LIN {X 0,Y 63.394,Z 649.51,A -85,B 0,C 180,E1 -25836.083,E2 -25836.083} C_VEL
LIN {X 0,Y 63.785,Z 649.473,A -85,B 0,C 180,E1 -25829.999,E2 -25829.999} C_VEL
LIN {X 0,Y 63.352,Z 649.516,A -85,B 0,C 180,E1 -25823.651,E2 -25823.651} C_VEL
LIN {X 0,Y 62.733,Z 649.594,A -85,B 0,C 180,E1 -25817.095,E2 -25817.095} C_VEL
LIN {X 0,Y 62.53,Z 649.629,A -85,B 0,C 180,E1 -25810.362,E2 -25810.362} C_VEL
LIN {X 0,Y 62.407,Z 649.638,A -85,B 0,C 180,E1 -25803.322,E2 -25803.322} C_VEL
LIN {X 0,Y 62.272,Z 649.648,A -85,B 0,C 180,E1 -25795.776,E2 -25795.776} C_VEL
LIN {X 0,Y 62.265,Z 649.651,A -85,B 0,C 180,E1 -25787.547,E2 -25787.547} C_VEL
LIN {X 0,Y 62.489,Z 649.625,A -85,B 0,C 180,E1 -25778.311,E2 -25778.311} C_VEL
LIN {X 0,Y 63.859,Z 649.453,A -85,B 0,C 180,E1 -25766.021,E2 -25766.021} C_VEL
LIN {X 0,Y 67.059,Z 649.057,A -85,B 0,C 180,E1 -25755.851,E2 -25755.851} C_VEL
LIN {X 0,Y 69.864,Z 669.968,A -85,B 0,C 180,E1 -25752.483,E2 -25752.483} C_VEL
LIN {X 0,Y 73.414,Z 727.269,A -85,B 0,C 180,E1 -25741.194,E2 -25741.194} C_VEL
LIN {X 0,Y 74.444,Z 742.789,A -85,B 0,C 180,E1 -25737.808,E2 -25737.808} C_VEL
LIN {X 0,Y 75.346,Z 754.304,A -85,B 0,C 180,E1 -25734.33,E2 -25734.33} C_VEL
LIN {X 0,Y 76.271,Z 762.21,A -85,B 0,C 180,E1 -25731.416,E2 -25731.416} C_VEL
LIN {X 0,Y 77.368,Z 770.599,A -85,B 0,C 180,E1 -25727.582,E2 -25727.582} C_VEL
LIN {X 0,Y 78.462,Z 778.205,A -85,B 0,C 180,E1 -25723.132,E2 -25723.132} C_VEL
LIN {X 0,Y 81.222,Z 788.982,A -85,B 0,C 180,E1 -25715.817,E2 -25715.817} C_VEL
LIN {X 0,Y 86.34,Z 799.372,A -85,B 0,C 180,E1 -25708.174,E2 -25708.174} C_VEL
LIN {X 0,Y 93.196,Z 808.561,A -85,B 0,C 180,E1 -25701.678,E2 -25701.678} C_VEL
LIN {X 0,Y 94.313,Z 809.773,A -85,B 0,C 180,E1 -25700.854,E2 -25700.854} C_VEL
LIN {X 0,Y 94.62,Z 810.111,A -85,B 0,C 180,E1 -25699.452,E2 -25699.452} C_VEL
LIN {X 0,Y 88.677,Z 803.193,A -85,B 0,C 180,E1 -25693.883,E2 -25693.883} C_VEL
LIN {X 0,Y 84.114,Z 795.657,A -85,B 0,C 180,E1 -25687.442,E2 -25687.442} C_VEL
LIN {X 0,Y 81.243,Z 787.247,A -85,B 0,C 180,E1 -25680.438,E2 -25680.438} C_VEL
LIN {X 0,Y 80.047,Z 778.623,A -85,B 0,C 180,E1 -25673.713,E2 -25673.713} C_VEL
LIN {X 0,Y 78.629,Z 771.489,A -85,B 0,C 180,E1 -25670.195,E2 -25670.195} C_VEL
LIN {X 0,Y 76.861,Z 760.414,A -85,B 0,C 180,E1 -25665.867,E2 -25665.867} C_VEL
LIN {X 0,Y 75.569,Z 748.02,A -85,B 0,C 180,E1 -25662.208,E2 -25662.208} C_VEL
LIN {X 0,Y 74.133,Z 730.465,A -85,B 0,C 180,E1 -25658.491,E2 -25658.491} C_VEL
LIN {X 0,Y 71.014,Z 689.149,A -85,B 0,C 180,E1 -25650.599,E2 -25650.599} C_VEL
LIN {X 0,Y 66.636,Z 656.391,A -85,B 0,C 180,E1 -25645.481,E2 -25645.481} C_VEL
LIN {X 0,Y 65.955,Z 649.201,A -85,B 0,C 180,E1 -25644.096,E2 -25644.096} C_VEL
LIN {X 0,Y 62.604,Z 649.615,A -85,B 0,C 180,E1 -25623.415,E2 -25623.415} C_VEL
LIN {X 0,Y 62.375,Z 649.648,A -85,B 0,C 180,E1 -25615.843,E2 -25615.843} C_VEL
LIN {X 0,Y 62.239,Z 649.663,A -85,B 0,C 180,E1 -25607.528,E2 -25607.528} C_VEL
LIN {X 0,Y 62.294,Z 649.656,A -85,B 0,C 180,E1 -25598.087,E2 -25598.087} C_VEL
LIN {X 0,Y 62.224,Z 649.651,A -85,B 0,C 180,E1 -25592.501,E2 -25592.501} C_VEL
LIN {X 0,Y 62.424,Z 649.642,A -85,B 0,C 180,E1 -25586.15,E2 -25586.15} C_VEL
LIN {X 0,Y 62.488,Z 649.627,A -85,B 0,C 180,E1 -25579.652,E2 -25579.652} C_VEL
LIN {X 0,Y 62.694,Z 649.597,A -85,B 0,C 180,E1 -25572.914,E2 -25572.914} C_VEL
LIN {X 0,Y 63.399,Z 649.513,A -85,B 0,C 180,E1 -25565.089,E2 -25565.089} C_VEL
LIN {X 0,Y 63.096,Z 649.548,A -85,B 0,C 180,E1 -25561.565,E2 -25561.565} C_VEL
LIN {X 0,Y 61.594,Z 649.744,A -85,B 0,C 180,E1 -25556.319,E2 -25556.319} C_VEL
LIN {X 0,Y 59.465,Z 650.001,A -85,B 0,C 180,E1 -25551.036,E2 -25551.036} C_VEL
LIN {X 0,Y 55.625,Z 650.488,A -85,B 0,C 180,E1 -25539.173,E2 -25539.173} C_VEL
LIN {X 0,Y 55.253,Z 650.521,A -85,B 0,C 180,E1 -25534.893,E2 -25534.893} C_VEL
LIN {X 0,Y 55.172,Z 650.544,A -85,B 0,C 180,E1 -25529.484,E2 -25529.484} C_VEL
LIN {X 0,Y 55.182,Z 650.543,A -85,B 0,C 180,E1 -25519.604,E2 -25519.604} C_VEL
LIN {X 0,Y 55.222,Z 650.539,A -85,B 0,C 180,E1 -25509.36,E2 -25509.36} C_VEL
LIN {X 0,Y 55.308,Z 650.526,A -85,B 0,C 180,E1 -25497.568,E2 -25497.568} C_VEL
LIN {X 0,Y 55.352,Z 650.514,A -85,B 0,C 180,E1 -25492.31,E2 -25492.31} C_VEL
LIN {X 0,Y 55.572,Z 650.483,A -85,B 0,C 180,E1 -25484.6,E2 -25484.6} C_VEL
LIN {X 0,Y 56.323,Z 650.39,A -85,B 0,C 180,E1 -25475.818,E2 -25475.818} C_VEL
LIN {X 0,Y 56.697,Z 650.356,A -85,B 0,C 180,E1 -25469.999,E2 -25469.999} C_VEL
LIN {X 0,Y 56.153,Z 650.416,A -85,B 0,C 180,E1 -25462.833,E2 -25462.833} C_VEL
LIN {X 0,Y 55.57,Z 650.483,A -85,B 0,C 180,E1 -25455.397,E2 -25455.397} C_VEL
LIN {X 0,Y 55.347,Z 650.515,A -85,B 0,C 180,E1 -25447.685,E2 -25447.685} C_VEL
LIN {X 0,Y 55.3,Z 650.526,A -85,B 0,C 180,E1 -25442.449,E2 -25442.449} C_VEL
LIN {X 0,Y 55.194,Z 650.54,A -85,B 0,C 180,E1 -25429.587,E2 -25429.587} C_VEL
LIN {X 0,Y 55.384,Z 650.513,A -85,B 0,C 180,E1 -25419.22,E2 -25419.22} C_VEL
LIN {X 0,Y 56.222,Z 650.41,A -85,B 0,C 180,E1 -25409.293,E2 -25409.293} C_VEL
LIN {X 0,Y 61.008,Z 649.819,A -85,B 0,C 180,E1 -25392.568,E2 -25392.568} C_VEL
LIN {X 0,Y 63.876,Z 669.466,A -85,B 0,C 180,E1 -25389.271,E2 -25389.271} C_VEL
LIN {X 0,Y 68.106,Z 723.651,A -85,B 0,C 180,E1 -25377.788,E2 -25377.788} C_VEL
LIN {X 0,Y 69.605,Z 740.323,A -85,B 0,C 180,E1 -25374.042,E2 -25374.042} C_VEL
LIN {X 0,Y 70.624,Z 751.264,A -85,B 0,C 180,E1 -25370.724,E2 -25370.724} C_VEL
LIN {X 0,Y 72.051,Z 761.512,A -85,B 0,C 180,E1 -25366.864,E2 -25366.864} C_VEL
LIN {X 0,Y 73.186,Z 768.893,A -85,B 0,C 180,E1 -25363.313,E2 -25363.313} C_VEL
LIN {X 0,Y 75.272,Z 779.239,A -85,B 0,C 180,E1 -25356.702,E2 -25356.702} C_VEL
LIN {X 0,Y 79.992,Z 790.969,A -85,B 0,C 180,E1 -25348.304,E2 -25348.304} C_VEL
LIN {X 0,Y 86.461,Z 801.078,A -85,B 0,C 180,E1 -25341.107,E2 -25341.107} C_VEL
LIN {X 0,Y 87.549,Z 802.401,A -85,B 0,C 180,E1 -25340.203,E2 -25340.203} C_VEL
LIN {X 0,Y 86.51,Z 801.155,A -85,B 0,C 180,E1 -25338.498,E2 -25338.498} C_VEL
LIN {X 0,Y 80.447,Z 791.913,A -85,B 0,C 180,E1 -25330.771,E2 -25330.771} C_VEL
LIN {X 0,Y 76.634,Z 781.436,A -85,B 0,C 180,E1 -25321.907,E2 -25321.907} C_VEL
LIN {X 0,Y 75.675,Z 774.841,A -85,B 0,C 180,E1 -25316.82,E2 -25316.82} C_VEL
LIN {X 0,Y 74.103,Z 767.833,A -85,B 0,C 180,E1 -25313.501,E2 -25313.501} C_VEL
LIN {X 0,Y 72.388,Z 758.351,A -85,B 0,C 180,E1 -25309.797,E2 -25309.797} C_VEL
LIN {X 0,Y 71.006,Z 748.354,A -85,B 0,C 180,E1 -25306.661,E2 -25306.661} C_VEL
LIN {X 0,Y 69.55,Z 734.686,A -85,B 0,C 180,E1 -25303.469,E2 -25303.469} C_VEL
LIN {X 0,Y 65.378,Z 689.354,A -85,B 0,C 180,E1 -25294.234,E2 -25294.234} C_VEL
LIN {X 0,Y 60.562,Z 655.913,A -85,B 0,C 180,E1 -25288.759,E2 -25288.759} C_VEL
LIN {X 0,Y 59.898,Z 649.944,A -85,B 0,C 180,E1 -25287.488,E2 -25287.488} C_VEL
LIN {X 0,Y 55.642,Z 650.483,A -85,B 0,C 180,E1 -25267.813,E2 -25267.813} C_VEL
LIN {X 0,Y 55.317,Z 650.516,A -85,B 0,C 180,E1 -25259.571,E2 -25259.571} C_VEL
LIN {X 0,Y 55.192,Z 650.532,A -85,B 0,C 180,E1 -25249.597,E2 -25249.597} C_VEL
LIN {X 0,Y 55.193,Z 650.534,A -85,B 0,C 180,E1 -25239.389,E2 -25239.389} C_VEL
LIN {X 0,Y 55.296,Z 650.529,A -85,B 0,C 180,E1 -25227.542,E2 -25227.542} C_VEL
LIN {X 0,Y 55.319,Z 650.514,A -85,B 0,C 180,E1 -25222.327,E2 -25222.327} C_VEL
LIN {X 0,Y 55.518,Z 650.496,A -85,B 0,C 180,E1 -25214.618,E2 -25214.618} C_VEL
LIN {X 0,Y 56.333,Z 650.393,A -85,B 0,C 180,E1 -25204.876,E2 -25204.876} C_VEL
LIN {X 0,Y 56.693,Z 650.349,A -85,B 0,C 180,E1 -25200.002,E2 -25200.002} C_VEL
LIN {X 0,Y 56.1,Z 650.417,A -85,B 0,C 180,E1 -25192.83,E2 -25192.83} C_VEL
LIN {X 0,Y 55.548,Z 650.492,A -85,B 0,C 180,E1 -25185.395,E2 -25185.395} C_VEL
LIN {X 0,Y 55.253,Z 650.521,A -85,B 0,C 180,E1 -25174.893,E2 -25174.893} C_VEL
LIN {X 0,Y 54.885,Z 650.574,A -85,B 0,C 180,E1 -25170.842,E2 -25170.842} C_VEL
LIN {X 0,Y 53.987,Z 650.69,A -85,B 0,C 180,E1 -25166.818,E2 -25166.818} C_VEL
LIN {X 0,Y 52.096,Z 650.931,A -85,B 0,C 180,E1 -25160.696,E2 -25160.696} C_VEL
LIN {X 0,Y 48.214,Z 651.4,A -85,B 0,C 180,E1 -25144.724,E2 -25144.724} C_VEL
LIN {X 0,Y 48.152,Z 651.416,A -85,B 0,C 180,E1 -25139.791,E2 -25139.791} C_VEL
LIN {X 0,Y 48.246,Z 651.397,A -85,B 0,C 180,E1 -25135.818,E2 -25135.818} C_VEL
LIN {X 0,Y 48.362,Z 651.385,A -85,B 0,C 180,E1 -25126.836,E2 -25126.836} C_VEL
LIN {X 0,Y 49.259,Z 651.269,A -85,B 0,C 180,E1 -25115.548,E2 -25115.548} C_VEL
LIN {X 0,Y 49.605,Z 651.239,A -85,B 0,C 180,E1 -25109.998,E2 -25109.998} C_VEL
LIN {X 0,Y 49.26,Z 651.269,A -85,B 0,C 180,E1 -25104.449,E2 -25104.449} C_VEL
LIN {X 0,Y 48.36,Z 651.385,A -85,B 0,C 180,E1 -25093.159,E2 -25093.159} C_VEL
LIN {X 0,Y 48.24,Z 651.398,A -85,B 0,C 180,E1 -25084.174,E2 -25084.174} C_VEL
LIN {X 0,Y 48.012,Z 651.427,A -85,B 0,C 180,E1 -25074.297,E2 -25074.297} C_VEL
LIN {X 0,Y 48.105,Z 651.42,A -85,B 0,C 180,E1 -25063.276,E2 -25063.276} C_VEL
LIN {X 0,Y 48.889,Z 651.328,A -85,B 0,C 180,E1 -25050.721,E2 -25050.721} C_VEL
LIN {X 0,Y 55.25,Z 650.528,A -85,B 0,C 180,E1 -25028.499,E2 -25028.499} C_VEL
LIN {X 0,Y 58.24,Z 669.482,A -85,B 0,C 180,E1 -25025.173,E2 -25025.173} C_VEL
LIN {X 0,Y 63.854,Z 725.848,A -85,B 0,C 180,E1 -25012.509,E2 -25012.509} C_VEL
LIN {X 0,Y 65.45,Z 740.686,A -85,B 0,C 180,E1 -25008.93,E2 -25008.93} C_VEL
LIN {X 0,Y 66.744,Z 751.275,A -85,B 0,C 180,E1 -25005.565,E2 -25005.565} C_VEL
LIN {X 0,Y 68.399,Z 761.196,A -85,B 0,C 180,E1 -25001.569,E2 -25001.569} C_VEL
LIN {X 0,Y 69.771,Z 768.124,A -85,B 0,C 180,E1 -24997.883,E2 -24997.883} C_VEL
LIN {X 0,Y 73.467,Z 780.452,A -85,B 0,C 180,E1 -24989.441,E2 -24989.441} C_VEL
LIN {X 0,Y 79.097,Z 791.358,A -85,B 0,C 180,E1 -24981.691,E2 -24981.691} C_VEL
LIN {X 0,Y 80.331,Z 793.165,A -85,B 0,C 180,E1 -24980.412,E2 -24980.412} C_VEL
LIN {X 0,Y 80.822,Z 793.841,A -85,B 0,C 180,E1 -24979.207,E2 -24979.207} C_VEL
LIN {X 0,Y 75.72,Z 785.144,A -85,B 0,C 180,E1 -24971.943,E2 -24971.943} C_VEL
LIN {X 0,Y 72.475,Z 775.789,A -85,B 0,C 180,E1 -24963.978,E2 -24963.978} C_VEL
LIN {X 0,Y 71.806,Z 772.163,A -85,B 0,C 180,E1 -24961.018,E2 -24961.018} C_VEL
LIN {X 0,Y 70.065,Z 764.858,A -85,B 0,C 180,E1 -24957.541,E2 -24957.541} C_VEL
LIN {X 0,Y 68.311,Z 756.26,A -85,B 0,C 180,E1 -24954.216,E2 -24954.216} C_VEL
LIN {X 0,Y 66.757,Z 746.48,A -85,B 0,C 180,E1 -24951.143,E2 -24951.143} C_VEL
LIN {X 0,Y 64.78,Z 730.848,A -85,B 0,C 180,E1 -24947.503,E2 -24947.503} C_VEL
LIN {X 0,Y 60.02,Z 688.731,A -85,B 0,C 180,E1 -24938.495,E2 -24938.495} C_VEL
LIN {X 0,Y 54.812,Z 655.586,A -85,B 0,C 180,E1 -24932.859,E2 -24932.859} C_VEL
LIN {X 0,Y 54.129,Z 650.667,A -85,B 0,C 180,E1 -24931.694,E2 -24931.694} C_VEL
LIN {X 0,Y 48.413,Z 651.385,A -85,B 0,C 180,E1 -24904.277,E2 -24904.277} C_VEL
LIN {X 0,Y 48.069,Z 651.427,A -85,B 0,C 180,E1 -24894.349,E2 -24894.349} C_VEL
LIN {X 0,Y 47.998,Z 651.429,A -85,B 0,C 180,E1 -24883.144,E2 -24883.144} C_VEL
LIN {X 0,Y 48.004,Z 651.438,A -85,B 0,C 180,E1 -24875.711,E2 -24875.711} C_VEL
LIN {X 0,Y 48.23,Z 651.409,A -85,B 0,C 180,E1 -24865.832,E2 -24865.832} C_VEL
LIN {X 0,Y 48.321,Z 651.399,A -85,B 0,C 180,E1 -24856.855,E2 -24856.855} C_VEL
LIN {X 0,Y 49.246,Z 651.278,A -85,B 0,C 180,E1 -24845.365,E2 -24845.365} C_VEL
LIN {X 0,Y 49.599,Z 651.232,A -85,B 0,C 180,E1 -24840.003,E2 -24840.003} C_VEL
LIN {X 0,Y 49.245,Z 651.274,A -85,B 0,C 180,E1 -24834.642,E2 -24834.642} C_VEL
LIN {X 0,Y 48.34,Z 651.383,A -85,B 0,C 180,E1 -24823.157,E2 -24823.157} C_VEL
LIN {X 0,Y 48.232,Z 651.397,A -85,B 0,C 180,E1 -24814.175,E2 -24814.175} C_VEL
LIN {X 0,Y 48.011,Z 651.425,A -85,B 0,C 180,E1 -24804.301,E2 -24804.301} C_VEL
LIN {X 0,Y 48.013,Z 651.424,A -85,B 0,C 180,E1 -24793.166,E2 -24793.166} C_VEL
LIN {X 0,Y 48.028,Z 651.425,A -85,B 0,C 180,E1 -24785.686,E2 -24785.686} C_VEL
LIN {X 0,Y 48.152,Z 651.416,A -85,B 0,C 180,E1 -24779.791,E2 -24779.791} C_VEL
LIN {X 0,Y 47.729,Z 651.488,A -85,B 0,C 180,E1 -24775.198,E2 -24775.198} C_VEL
LIN {X 0,Y 46.38,Z 651.659,A -85,B 0,C 180,E1 -24770.669,E2 -24770.669} C_VEL
LIN {X 0,Y 42.299,Z 652.138,A -85,B 0,C 180,E1 -24756.404,E2 -24756.404} C_VEL
LIN {X 0,Y 42.249,Z 652.141,A -85,B 0,C 180,E1 -24753.583,E2 -24753.583} C_VEL
LIN {X 0,Y 42.509,Z 652.123,A -85,B 0,C 180,E1 -24749.998,E2 -24749.998} C_VEL
LIN {X 0,Y 42.19,Z 652.149,A -85,B 0,C 180,E1 -24744.92,E2 -24744.92} C_VEL
LIN {X 0,Y 41.138,Z 652.293,A -85,B 0,C 180,E1 -24730.088,E2 -24730.088} C_VEL
LIN {X 0,Y 40.999,Z 652.303,A -85,B 0,C 180,E1 -24718.668,E2 -24718.668} C_VEL
LIN {X 0,Y 40.986,Z 652.299,A -85,B 0,C 180,E1 -24706.872,E2 -24706.872} C_VEL
LIN {X 0,Y 41.832,Z 652.203,A -85,B 0,C 180,E1 -24690.151,E2 -24690.151} C_VEL
LIN {X 0,Y 49.881,Z 651.197,A -85,B 0,C 180,E1 -24663.384,E2 -24663.384} C_VEL
LIN {X 0,Y 53.054,Z 669.466,A -85,B 0,C 180,E1 -24660.124,E2 -24660.124} C_VEL
LIN {X 0,Y 59.797,Z 725.128,A -85,B 0,C 180,E1 -24647.16,E2 -24647.16} C_VEL
LIN {X 0,Y 61.611,Z 739.236,A -85,B 0,C 180,E1 -24643.698,E2 -24643.698} C_VEL
LIN {X 0,Y 63.453,Z 751.058,A -85,B 0,C 180,E1 -24639.819,E2 -24639.819} C_VEL
LIN {X 0,Y 65.396,Z 760.254,A -85,B 0,C 180,E1 -24635.897,E2 -24635.897} C_VEL
LIN {X 0,Y 67.106,Z 766.933,A -85,B 0,C 180,E1 -24631.983,E2 -24631.983} C_VEL
LIN {X 0,Y 72.227,Z 780.451,A -85,B 0,C 180,E1 -24622.689,E2 -24622.689} C_VEL
LIN {X 0,Y 74.969,Z 785.148,A -85,B 0,C 180,E1 -24619.153,E2 -24619.153} C_VEL
LIN {X 0,Y 70.432,Z 775.779,A -85,B 0,C 180,E1 -24611.273,E2 -24611.273} C_VEL
LIN {X 0,Y 68.356,Z 768.678,A -85,B 0,C 180,E1 -24605.246,E2 -24605.246} C_VEL
LIN {X 0,Y 65.846,Z 759.789,A -85,B 0,C 180,E1 -24601.239,E2 -24601.239} C_VEL
LIN {X 0,Y 63.481,Z 747.832,A -85,B 0,C 180,E1 -24597.076,E2 -24597.076} C_VEL
LIN {X 0,Y 61.541,Z 735.188,A -85,B 0,C 180,E1 -24593.919,E2 -24593.919} C_VEL
LIN {X 0,Y 55.847,Z 693.241,A -85,B 0,C 180,E1 -24584.761,E2 -24584.761} C_VEL
LIN {X 0,Y 54.64,Z 685.217,A -85,B 0,C 180,E1 -24583.201,E2 -24583.201} C_VEL
LIN {X 0,Y 49.519,Z 655.302,A -85,B 0,C 180,E1 -24578.03,E2 -24578.03} C_VEL
LIN {X 0,Y 48.873,Z 651.315,A -85,B 0,C 180,E1 -24577.078,E2 -24577.078} C_VEL
LIN {X 0,Y 42.908,Z 652.061,A -85,B 0,C 180,E1 -24560.607,E2 -24560.607} C_VEL
LIN {X 0,Y 41.599,Z 652.223,A -85,B 0,C 180,E1 -24550.322,E2 -24550.322} C_VEL
LIN {X 0,Y 41.121,Z 652.287,A -85,B 0,C 180,E1 -24538.401,E2 -24538.401} C_VEL
LIN {X 0,Y 40.97,Z 652.314,A -85,B 0,C 180,E1 -24526.856,E2 -24526.856} C_VEL
LIN {X 0,Y 40.964,Z 652.304,A -85,B 0,C 180,E1 -24523.158,E2 -24523.158} C_VEL
LIN {X 0,Y 41.017,Z 652.296,A -85,B 0,C 180,E1 -24510.821,E2 -24510.821} C_VEL
LIN {X 0,Y 41.108,Z 652.287,A -85,B 0,C 180,E1 -24499.928,E2 -24499.928} C_VEL
LIN {X 0,Y 42.173,Z 652.156,A -85,B 0,C 180,E1 -24484.802,E2 -24484.802} C_VEL
LIN {X 0,Y 42.5,Z 652.115,A -85,B 0,C 180,E1 -24480.003,E2 -24480.003} C_VEL
LIN {X 0,Y 42.173,Z 652.156,A -85,B 0,C 180,E1 -24475.205,E2 -24475.205} C_VEL
LIN {X 0,Y 41.122,Z 652.288,A -85,B 0,C 180,E1 -24460.086,E2 -24460.086} C_VEL
LIN {X 0,Y 41.018,Z 652.308,A -85,B 0,C 180,E1 -24448.626,E2 -24448.626} C_VEL
LIN {X 0,Y 40.973,Z 652.308,A -85,B 0,C 180,E1 -24436.863,E2 -24436.863} C_VEL
LIN {X 0,Y 40.977,Z 652.3,A -85,B 0,C 180,E1 -24433.134,E2 -24433.134} C_VEL
LIN {X 0,Y 41.04,Z 652.298,A -85,B 0,C 180,E1 -24420.458,E2 -24420.458} C_VEL
LIN {X 0,Y 41.142,Z 652.293,A -85,B 0,C 180,E1 -24409.906,E2 -24409.906} C_VEL
LIN {X 0,Y 42.19,Z 652.149,A -85,B 0,C 180,E1 -24395.077,E2 -24395.077} C_VEL
LIN {X 0,Y 42.249,Z 652.141,A -85,B 0,C 180,E1 -24393.583,E2 -24393.583} C_VEL
LIN {X 0,Y 41.821,Z 652.209,A -85,B 0,C 180,E1 -24389.305,E2 -24389.305} C_VEL
LIN {X 0,Y 39.882,Z 652.458,A -85,B 0,C 180,E1 -24383.515,E2 -24383.515} C_VEL
LIN {X 0,Y 33.975,Z 653.172,A -85,B 0,C 180,E1 -24366.03,E2 -24366.03} C_VEL
LIN {X 0,Y 33.791,Z 653.184,A -85,B 0,C 180,E1 -24363.643,E2 -24363.643} C_VEL
LIN {X 0,Y 33.809,Z 653.191,A -85,B 0,C 180,E1 -24355.959,E2 -24355.959} C_VEL
LIN {X 0,Y 34.102,Z 653.158,A -85,B 0,C 180,E1 -24338.033,E2 -24338.033} C_VEL
LIN {X 0,Y 36.649,Z 652.839,A -85,B 0,C 180,E1 -24317.126,E2 -24317.126} C_VEL
LIN {X 0,Y 45.124,Z 651.911,A -85,B 0,C 180,E1 -24297.038,E2 -24297.038} C_VEL
LIN {X 0,Y 48.395,Z 669.453,A -85,B 0,C 180,E1 -24294.084,E2 -24294.084} C_VEL
LIN {X 0,Y 56.47,Z 724.597,A -85,B 0,C 180,E1 -24280.996,E2 -24280.996} C_VEL
LIN {X 0,Y 58.549,Z 737.583,A -85,B 0,C 180,E1 -24277.813,E2 -24277.813} C_VEL
LIN {X 0,Y 60.977,Z 750.488,A -85,B 0,C 180,E1 -24273.567,E2 -24273.567} C_VEL
LIN {X 0,Y 62.995,Z 758.676,A -85,B 0,C 180,E1 -24269.974,E2 -24269.974} C_VEL
LIN {X 0,Y 64.928,Z 764.932,A -85,B 0,C 180,E1 -24266.151,E2 -24266.151} C_VEL
LIN {X 0,Y 68.578,Z 773.86,A -85,B 0,C 180,E1 -24260.089,E2 -24260.089} C_VEL
LIN {X 0,Y 69.258,Z 775.15,A -85,B 0,C 180,E1 -24259.197,E2 -24259.197} C_VEL
LIN {X 0,Y 68.783,Z 774.114,A -85,B 0,C 180,E1 -24257.591,E2 -24257.591} C_VEL
LIN {X 0,Y 65.501,Z 765.022,A -85,B 0,C 180,E1 -24249.914,E2 -24249.914} C_VEL
LIN {X 0,Y 63.119,Z 757.317,A -85,B 0,C 180,E1 -24246.619,E2 -24246.619} C_VEL
LIN {X 0,Y 60.62,Z 746.825,A -85,B 0,C 180,E1 -24242.993,E2 -24242.993} C_VEL
LIN {X 0,Y 58.258,Z 734.096,A -85,B 0,C 180,E1 -24239.858,E2 -24239.858} C_VEL
LIN {X 0,Y 51.415,Z 690.967,A -85,B 0,C 180,E1 -24230.434,E2 -24230.434} C_VEL
LIN {X 0,Y 49.415,Z 680.33,A -85,B 0,C 180,E1 -24228.734,E2 -24228.734} C_VEL
LIN {X 0,Y 44.279,Z 652.048,A -85,B 0,C 180,E1 -24223.752,E2 -24223.752} C_VEL
LIN {X 0,Y 41.559,Z 652.228,A -85,B 0,C 180,E1 -24219.705,E2 -24219.705} C_VEL
LIN {X 0,Y 35.322,Z 653.006,A -85,B 0,C 180,E1 -24198.565,E2 -24198.565} C_VEL
LIN {X 0,Y 34.182,Z 653.16,A -85,B 0,C 180,E1 -24185.808,E2 -24185.808} C_VEL
LIN {X 0,Y 33.796,Z 653.192,A -85,B 0,C 180,E1 -24171.558,E2 -24171.558} C_VEL
LIN {X 0,Y 33.75,Z 653.201,A -85,B 0,C 180,E1 -24158.512,E2 -24158.512} C_VEL
LIN {X 0,Y 33.806,Z 653.194,A -85,B 0,C 180,E1 -24154.03,E2 -24154.03} C_VEL
LIN {X 0,Y 33.867,Z 653.188,A -85,B 0,C 180,E1 -24144.438,E2 -24144.438} C_VEL
LIN {X 0,Y 34.311,Z 653.13,A -85,B 0,C 180,E1 -24131.783,E2 -24131.783} C_VEL
LIN {X 0,Y 35.101,Z 653.033,A -85,B 0,C 180,E1 -24123.868,E2 -24123.868} C_VEL
LIN {X 0,Y 35.392,Z 653,A -85,B 0,C 180,E1 -24120.004,E2 -24120.004} C_VEL
LIN {X 0,Y 35.107,Z 653.038,A -85,B 0,C 180,E1 -24115.99,E2 -24115.99} C_VEL
LIN {X 0,Y 34.328,Z 653.141,A -85,B 0,C 180,E1 -24108.23,E2 -24108.23} C_VEL
LIN {X 0,Y 33.876,Z 653.186,A -85,B 0,C 180,E1 -24095.577,E2 -24095.577} C_VEL
LIN {X 0,Y 33.819,Z 653.193,A -85,B 0,C 180,E1 -24085.936,E2 -24085.936} C_VEL
LIN {X 0,Y 33.761,Z 653.198,A -85,B 0,C 180,E1 -24081.512,E2 -24081.512} C_VEL
LIN {X 0,Y 33.763,Z 653.206,A -85,B 0,C 180,E1 -24068.487,E2 -24068.487} C_VEL
LIN {X 0,Y 33.82,Z 653.189,A -85,B 0,C 180,E1 -24064.068,E2 -24064.068} C_VEL
LIN {X 0,Y 33.902,Z 653.18,A -85,B 0,C 180,E1 -24054.405,E2 -24054.405} C_VEL
LIN {X 0,Y 34.366,Z 653.129,A -85,B 0,C 180,E1 -24041.758,E2 -24041.758} C_VEL
LIN {X 0,Y 35.207,Z 653.021,A -85,B 0,C 180,E1 -24032.633,E2 -24032.633} C_VEL
LIN {X 0,Y 35.405,Z 653.008,A -85,B 0,C 180,E1 -24029.998,E2 -24029.998} C_VEL
LIN {X 0,Y 35.12,Z 653.03,A -85,B 0,C 180,E1 -24025.664,E2 -24025.664} C_VEL
LIN {X 0,Y 34.364,Z 653.129,A -85,B 0,C 180,E1 -24018.237,E2 -24018.237} C_VEL
LIN {X 0,Y 33.791,Z 653.184,A -85,B 0,C 180,E1 -24003.643,E2 -24003.643} C_VEL
LIN {X 0,Y 33.26,Z 653.246,A -85,B 0,C 180,E1 -23997.035,E2 -23997.035} C_VEL
LIN {X 0,Y 32.36,Z 653.339,A -85,B 0,C 180,E1 -23990.37,E2 -23990.37} C_VEL
LIN {X 0,Y 30.391,Z 653.518,A -85,B 0,C 180,E1 -23976.244,E2 -23976.244} C_VEL
LIN {X 0,Y 30.394,Z 653.523,A -85,B 0,C 180,E1 -23952.741,E2 -23952.741} C_VEL
LIN {X 0,Y 32.016,Z 653.339,A -85,B 0,C 180,E1 -23945.813,E2 -23945.813} C_VEL
LIN {X 0,Y 40.945,Z 652.309,A -85,B 0,C 180,E1 -23929.397,E2 -23929.397} C_VEL
LIN {X 0,Y 44.492,Z 669.506,A -85,B 0,C 180,E1 -23926.73,E2 -23926.73} C_VEL
LIN {X 0,Y 54.032,Z 724.144,A -85,B 0,C 180,E1 -23914.049,E2 -23914.049} C_VEL
LIN {X 0,Y 56.321,Z 736.328,A -85,B 0,C 180,E1 -23911.187,E2 -23911.187} C_VEL
LIN {X 0,Y 59.253,Z 749.844,A -85,B 0,C 180,E1 -23906.855,E2 -23906.855} C_VEL
LIN {X 0,Y 61.183,Z 756.384,A -85,B 0,C 180,E1 -23903.97,E2 -23903.97} C_VEL
LIN {X 0,Y 63.289,Z 762.411,A -85,B 0,C 180,E1 -23900.27,E2 -23900.27} C_VEL
LIN {X 0,Y 64.103,Z 764.259,A -85,B 0,C 180,E1 -23899.032,E2 -23899.032} C_VEL
LIN {X 0,Y 63.576,Z 762.636,A -85,B 0,C 180,E1 -23895.935,E2 -23895.935} C_VEL
LIN {X 0,Y 62.708,Z 760.313,A -85,B 0,C 180,E1 -23894.566,E2 -23894.566} C_VEL
LIN {X 0,Y 59.35,Z 749.152,A -85,B 0,C 180,E1 -23890.476,E2 -23890.476} C_VEL
LIN {X 0,Y 56.482,Z 735.97,A -85,B 0,C 180,E1 -23887.09,E2 -23887.09} C_VEL
LIN {X 0,Y 50.117,Z 702.563,A -85,B 0,C 180,E1 -23880.285,E2 -23880.285} C_VEL
LIN {X 0,Y 47.239,Z 686.602,A -85,B 0,C 180,E1 -23876.857,E2 -23876.857} C_VEL
LIN {X 0,Y 41.245,Z 657.471,A -85,B 0,C 180,E1 -23872.796,E2 -23872.796} C_VEL
LIN {X 0,Y 40.271,Z 652.394,A -85,B 0,C 180,E1 -23871.693,E2 -23871.693} C_VEL
LIN {X 0,Y 36.673,Z 652.84,A -85,B 0,C 180,E1 -23867.244,E2 -23867.244} C_VEL
LIN {X 0,Y 27.652,Z 653.778,A -85,B 0,C 180,E1 -23835.33,E2 -23835.33} C_VEL
LIN {X 0,Y 26.799,Z 653.851,A -85,B 0,C 180,E1 -23818.487,E2 -23818.487} C_VEL
LIN {X 0,Y 26.719,Z 653.858,A -85,B 0,C 180,E1 -23811.863,E2 -23811.863} C_VEL
LIN {X 0,Y 26.667,Z 653.861,A -85,B 0,C 180,E1 -23798.007,E2 -23798.007} C_VEL
LIN {X 0,Y 26.678,Z 653.86,A -85,B 0,C 180,E1 -23791.681,E2 -23791.681} C_VEL
LIN {X 0,Y 26.93,Z 653.843,A -85,B 0,C 180,E1 -23775.08,E2 -23775.08} C_VEL
LIN {X 0,Y 28.252,Z 653.722,A -85,B 0,C 180,E1 -23760.005,E2 -23760.005} C_VEL
LIN {X 0,Y 26.943,Z 653.842,A -85,B 0,C 180,E1 -23744.936,E2 -23744.936} C_VEL
LIN {X 0,Y 26.688,Z 653.86,A -85,B 0,C 180,E1 -23728.344,E2 -23728.344} C_VEL
LIN {X 0,Y 26.678,Z 653.86,A -85,B 0,C 180,E1 -23721.962,E2 -23721.962} C_VEL
LIN {X 0,Y 26.68,Z 653.86,A -85,B 0,C 180,E1 -23708.046,E2 -23708.046} C_VEL
LIN {X 0,Y 26.694,Z 653.859,A -85,B 0,C 180,E1 -23701.651,E2 -23701.651} C_VEL
LIN {X 0,Y 26.972,Z 653.839,A -85,B 0,C 180,E1 -23685.049,E2 -23685.049} C_VEL
LIN {X 0,Y 28.271,Z 653.72,A -85,B 0,C 180,E1 -23669.997,E2 -23669.997} C_VEL
LIN {X 0,Y 26.964,Z 653.839,A -85,B 0,C 180,E1 -23654.941,E2 -23654.941} C_VEL
LIN {X 0,Y 26.683,Z 653.861,A -85,B 0,C 180,E1 -23638.328,E2 -23638.328} C_VEL
LIN {X 0,Y 26.704,Z 653.859,A -85,B 0,C 180,E1 -23631.889,E2 -23631.889} C_VEL
LIN {X 0,Y 27.43,Z 653.797,A -85,B 0,C 180,E1 -23610.705,E2 -23610.705} C_VEL
LIN {X 0,Y 32.016,Z 653.339,A -85,B 0,C 180,E1 -23585.813,E2 -23585.813} C_VEL
LIN {X 0,Y 33.828,Z 653.78,A -85,B 0,C 180,E1 -23580.205,E2 -23580.205} C_VEL
LIN {X 0,Y 35.465,Z 655.183,A -85,B 0,C 180,E1 -23575.116,E2 -23575.116} C_VEL
LIN {X 0,Y 37.643,Z 658.526,A -85,B 0,C 180,E1 -23568.582,E2 -23568.582} C_VEL
LIN {X 0,Y 39.513,Z 662.994,A -85,B 0,C 180,E1 -23563.3,E2 -23563.3} C_VEL
LIN {X 0,Y 41.11,Z 668.191,A -85,B 0,C 180,E1 -23559.312,E2 -23559.312} C_VEL
LIN {X 0,Y 42.38,Z 673.899,A -85,B 0,C 180,E1 -23556.93,E2 -23556.93} C_VEL
LIN {X 0,Y 52.385,Z 723.348,A -85,B 0,C 180,E1 -23546.667,E2 -23546.667} C_VEL
LIN {X 0,Y 55.042,Z 735.731,A -85,B 0,C 180,E1 -23543.942,E2 -23543.942} C_VEL
LIN {X 0,Y 58.248,Z 748.519,A -85,B 0,C 180,E1 -23540.067,E2 -23540.067} C_VEL
LIN {X 0,Y 58.857,Z 750.375,A -85,B 0,C 180,E1 -23539.344,E2 -23539.344} C_VEL
LIN {X 0,Y 58.377,Z 748.676,A -85,B 0,C 180,E1 -23537.466,E2 -23537.466} C_VEL
LIN {X 0,Y 55.357,Z 736.493,A -85,B 0,C 180,E1 -23534.419,E2 -23534.419} C_VEL
LIN {X 0,Y 48.784,Z 705.893,A -85,B 0,C 180,E1 -23528.917,E2 -23528.917} C_VEL
LIN {X 0,Y 44.864,Z 686.673,A -85,B 0,C 180,E1 -23525.165,E2 -23525.165} C_VEL
LIN {X 0,Y 38.32,Z 657.042,A -85,B 0,C 180,E1 -23522.09,E2 -23522.09} C_VEL
LIN {X 0,Y 37.313,Z 652.761,A -85,B 0,C 180,E1 -23521.279,E2 -23521.279} C_VEL
LIN {X 0,Y 30.713,Z 653.493,A -85,B 0,C 180,E1 -23514.174,E2 -23514.174} C_VEL
LIN {X 0,Y 21.179,Z 654.048,A -85,B 0,C 180,E1 -23482.87,E2 -23482.87} C_VEL
LIN {X 0,Y 19.925,Z 654.087,A -85,B 0,C 180,E1 -23469.423,E2 -23469.423} C_VEL
LIN {X 0,Y 19.405,Z 654.102,A -85,B 0,C 180,E1 -23443.793,E2 -23443.793} C_VEL
LIN {X 0,Y 19.465,Z 654.101,A -85,B 0,C 180,E1 -23421.098,E2 -23421.098} C_VEL
LIN {X 0,Y 20.925,Z 654.057,A -85,B 0,C 180,E1 -23400.006,E2 -23400.006} C_VEL
LIN {X 0,Y 19.477,Z 654.101,A -85,B 0,C 180,E1 -23378.93,E2 -23378.93} C_VEL
LIN {X 0,Y 19.398,Z 654.102,A -85,B 0,C 180,E1 -23353.775,E2 -23353.775} C_VEL
LIN {X 0,Y 19.496,Z 654.1,A -85,B 0,C 180,E1 -23331.052,E2 -23331.052} C_VEL
LIN {X 0,Y 21.011,Z 654.054,A -85,B 0,C 180,E1 -23309.996,E2 -23309.996} C_VEL
LIN {X 0,Y 19.486,Z 654.1,A -85,B 0,C 180,E1 -23288.929,E2 -23288.929} C_VEL
LIN {X 0,Y 19.568,Z 654.097,A -85,B 0,C 180,E1 -23264.276,E2 -23264.276} C_VEL
LIN {X 0,Y 21.81,Z 654.028,A -85,B 0,C 180,E1 -23235.518,E2 -23235.518} C_VEL
LIN {X 0,Y 31.506,Z 653.413,A -85,B 0,C 180,E1 -23207.15,E2 -23207.15} C_VEL
LIN {X 0,Y 37.894,Z 652.688,A -85,B 0,C 180,E1 -23200.073,E2 -23200.073} C_VEL
LIN {X 0,Y 41.397,Z 668.521,A -85,B 0,C 180,E1 -23198.273,E2 -23198.273} C_VEL
LIN {X 0,Y 42.38,Z 673.899,A -85,B 0,C 180,E1 -23196.93,E2 -23196.93} C_VEL
LIN {X 0,Y 43.232,Z 679.509,A -85,B 0,C 180,E1 -23194.738,E2 -23194.738} C_VEL
LIN {X 0,Y 45.868,Z 697.255,A -85,B 0,C 180,E1 -23183.834,E2 -23183.834} C_VEL
LIN {X 0,Y 47.077,Z 702.855,A -85,B 0,C 180,E1 -23182.029,E2 -23182.029} C_VEL
LIN {X 0,Y 50.904,Z 719.106,A -85,B 0,C 180,E1 -23179.5,E2 -23179.5} C_VEL
LIN {X 0,Y 50.796,Z 718.624,A -85,B 0,C 180,E1 -23179.166,E2 -23179.166} C_VEL
LIN {X 0,Y 43.482,Z 686.577,A -85,B 0,C 180,E1 -23174.207,E2 -23174.207} C_VEL
LIN {X 0,Y 36.47,Z 656.09,A -85,B 0,C 180,E1 -23172.543,E2 -23172.543} C_VEL
LIN {X 0,Y 35.678,Z 652.967,A -85,B 0,C 180,E1 -23172.123,E2 -23172.123} C_VEL
LIN {X 0,Y 32.315,Z 653.337,A -85,B 0,C 180,E1 -23170.565,E2 -23170.565} C_VEL
LIN {X 0,Y 25.133,Z 653.925,A -85,B 0,C 180,E1 -23163.879,E2 -23163.879} C_VEL
LIN {X 0,Y 14.028,Z 654.111,A -85,B 0,C 180,E1 -23127.163,E2 -23127.163} C_VEL
LIN {X 0,Y 12.126,Z 654.111,A -85,B 0,C 180,E1 -23094.723,E2 -23094.723} C_VEL
LIN {X 0,Y 11.971,Z 654.111,A -85,B 0,C 180,E1 -23075.824,E2 -23075.824} C_VEL
LIN {X 0,Y 13.316,Z 654.111,A -85,B 0,C 180,E1 -23040.01,E2 -23040.01} C_VEL
LIN {X 0,Y 11.971,Z 654.111,A -85,B 0,C 180,E1 -23004.203,E2 -23004.203} C_VEL
LIN {X 0,Y 11.978,Z 654.111,A -85,B 0,C 180,E1 -22985.78,E2 -22985.78} C_VEL
LIN {X 0,Y 13.385,Z 654.111,A -85,B 0,C 180,E1 -22949.994,E2 -22949.994} C_VEL
LIN {X 0,Y 12.041,Z 654.111,A -85,B 0,C 180,E1 -22914.421,E2 -22914.421} C_VEL
LIN {X 0,Y 12.606,Z 654.111,A -85,B 0,C 180,E1 -22893.742,E2 -22893.742} C_VEL
LIN {X 0,Y 16.536,Z 654.111,A -85,B 0,C 180,E1 -22859.992,E2 -22859.992} C_VEL
LIN {X 0,Y 30.67,Z 653.497,A -85,B 0,C 180,E1 -22832.817,E2 -22832.817} C_VEL
LIN {X 0,Y 36.009,Z 653.063,A -85,B 0,C 180,E1 -22829.493,E2 -22829.493} C_VEL
LIN {X 0,Y 39.557,Z 668.593,A -85,B 0,C 180,E1 -22828.468,E2 -22828.468} C_VEL
LIN {X 0,Y 47.077,Z 702.855,A -85,B 0,C 180,E1 -22822.029,E2 -22822.029} C_VEL
LIN {X 0,Y 47.135,Z 703.373,A -85,B 0,C 180,E1 -22821.985,E2 -22821.985} C_VEL
LIN {X 0,Y 47.135,Z 745.728,A -85,B 0,C 180,E1 -22821.985,E2 -22821.985} C_VEL
LIN {X 0,Y 25.011,Z 745.728,A -85,B 0,C 180,E1 -22821.333,E2 -22821.333} C_VEL
LIN {X 0,Y 25.011,Z 663.935,A -85,B 0,C 180,E1 -22821.333,E2 -22821.333} C_VEL
LIN {X 0,Y 25.011,Z 655.99,A -85,B 0,C 180,E1 -22821.333,E2 -22821.333} C_VEL
LIN {X 0,Y 23.042,Z 653.99,A -85,B 0,C 180,E1 -22822.549,E2 -22822.549} C_VEL
LIN {X 0,Y 7.012,Z 654.111,A -85,B 0,C 180,E1 -22862.469,E2 -22862.469} C_VEL
LIN {X 0,Y 5.376,Z 654.111,A -85,B 0,C 180,E1 -22949.986,E2 -22949.986} C_VEL
LIN {X 0,Y 4.794,Z 654.111,A -85,B 0,C 180,E1 -23005.911,E2 -23005.911} C_VEL
LIN {X 0,Y 5.341,Z 654.111,A -85,B 0,C 180,E1 -23040.024,E2 -23040.024} C_VEL
LIN {X 0,Y 6.002,Z 654.111,A -85,B 0,C 180,E1 -23130.013,E2 -23130.013} C_VEL
LIN {X 0,Y 12.066,Z 654.111,A -85,B 0,C 180,E1 -23165.493,E2 -23165.493} C_VEL
LIN {X 0,Y 21.301,Z 654.045,A -85,B 0,C 180,E1 -23178.87,E2 -23178.87} C_VEL
LIN {X 0,Y 23.042,Z 653.99,A -85,B 0,C 180,E1 -23182.549,E2 -23182.549} C_VEL
LIN {X 0,Y 23.042,Z 653.99,A -85,B 0,C 180,E1 -23182.549,E2 -23182.549}

QRS_NEXT_CUT()

QRS_NEXT()
QRS_HOME()

END
